FUNCTION_BLOCK FB_TON_LTIME (* standard timer function block (on-delay timing) (LTIME) *)
  (* Standard: 61131-3; Classification: standard timer function block; Description: Copyright (c) 2011 TU Wien ACIN, Patrick Aigner, HR Agrartechnik GmbH This program and the accompanying materials are made available under the terms of the Eclipse Public License 2.0 which is available at https://www.eclipse.org/legal/epl-2.0/ SPDX-License-Identifier: EPL-2.0 Some portions generated by Gemini CLI *)
  (* Version 1.0, 2026-02-01, Franz Höpfinger, HR Agrartechnik GmbH, Copy over from FB_TON and made this Block *)
  PACKAGE iec61131::timers;
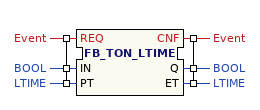
  EVENT_INPUT
    REQ WITH IN, PT; (* Normal Execution Request *)
  END_EVENT
  EVENT_OUTPUT
    CNF WITH Q, ET; (* Execution Confirmation *)
  END_EVENT
  VAR_INPUT
    IN : BOOL; (* Input *)
    PT : LTIME; (* Process time *)
  END_VAR
  VAR_OUTPUT
    Q : BOOL; (* Output *)
    ET : LTIME; (* Elapsed time *)
  END_VAR
  VAR
    MEM : BOOL; (* internal variable *)
    StartTime : LTIME; (* internal variable *)
  END_VAR
  EC_STATES
    REQ : REQ -> CNF;
  END_STATES
  ALGORITHM REQ IN ST:
VAR_TEMP
	SysTime : TIME;
END_VAR

SysTime := NOW_MONOTONIC();

IF NOT IN THEN
	Q := FALSE;
	ET := LT#0s;
	MEM := FALSE;
ELSE
	IF NOT MEM THEN
		StartTime := SysTime;
		MEM := TRUE;
	END_IF;

	IF NOT Q THEN
		ET := SysTime - StartTime;

		IF ET >= PT THEN
			ET := PT;
			Q := TRUE;
		END_IF;
	END_IF;
END_IF;
  END_ALGORITHM
END_FUNCTION_BLOCK
